FUNCTION_BLOCK PresenceDetector
VAR_INPUT
END_VAR
VAR_OUTPUT
	bAllPartsPresent : BOOL;
END_VAR
VAR
	aSensors : ARRAY[1..3] OF Sensor;
	fbTimer : TON;
	i: INT;
END_VAR

aSensors[1]();
aSensors[2]();
aSensors[3]();
fbTimer(
	IN:= aSensors[1].bSignal
		AND aSensors[2].bSignal
		AND aSensors[3].bSignal,
	PT:=T#2S
);
IF fbTimer.Q
THEN
	bAllPartsPresent := TRUE;
ELSE
	bAllPartsPresent :=FALSE;
END_IF

END_FUNCTION_BLOCK

(* stored: Version 1.1.0.1, ProductVersion 3.1.4024.2
   POU PresenceDetector: Id {6471a446-9fc3-4a13-92bb-00f1ae10de61}, SpecialFunc None *)
